// TIA Portal project "Supervisorios2" (V17)

(* hardware
DEVICE "S7-1200 station_1"  S7-1200 Station
   slot 0: "Rack_0"  S7-1200 Rack  Rack  V1.0
   slot 1: "PLC_1"  CPU 1212C AC/DC/Rly  6ES7 212-1BE40-0XB0  V4.4
   slot 2: "DI 8x24VDC_1"  6ES7 221-1BF32-0XB0  V2.0
   slot 3: "AQ 1x12BIT_1"  AQ1 signal board  6ES7 232-4HA30-0XB0  V1.0
DEVICE "HMI_1"  TP700 Comfort
   slot 0: "HMI_1"  TP700 Comfort  6AV2 124-0GC01-0AX0  17.0.0.0
   slot 1: "HMI_RT_1"  TP700 Comfort  6AV2 124-0GC01-0AX0  17.0.0.0
   slot 5: "HMI_1.IE_CP_1"  PROFINET Interface  17.0.0.0
      slot 1: "PROFINET Interface_1"  PROFINET Interface
         slot 1: "Port_1"  Port
         slot 2: "Port_2"  Port
   slot 7: "HMI_1.MPI/DP_CP_1"  MPI/DP Interface  17.0.0.0
*)

// ===== PLC "PLC_1"  CPU 1212C AC/DC/Rly =====

VAR_GLOBAL   // PLC tag table "Default tag table"
   "MemLED" AT %M32.0 : Bool;
   "MemL" AT %M32.1 : Bool;
   "norm" AT %MD8 : Real;
   "scal" AT %MD12 : Real;
   "potenciometro" AT %IW64 : Word;
   "SAIDA" AT %QD2 : Real;
   "Tag_2" AT %M101.2 : Bool;
   "Clock_Byte" AT %MB0 : Byte;
   "Clock_10Hz" AT %M0.0 : Bool;
   "Clock_5Hz" AT %M0.1 : Bool;
   "Clock_2.5Hz" AT %M0.2 : Bool;
   "Clock_2Hz" AT %M0.3 : Bool;
   "Clock_1.25Hz" AT %M0.4 : Bool;
   "Clock_1Hz" AT %M0.5 : Bool;
   "Clock_0.625Hz" AT %M0.6 : Bool;
   "Clock_0.5Hz" AT %M0.7 : Bool;
END_VAR

VAR_GLOBAL   // PLC tag table "ComportamentoRipas"
   "ON" AT %I0.0 : Bool;
   "OFF" AT %I0.1 : Bool;
   "S1" AT %I0.2 : Bool;
   "S2" AT %I0.3 : Bool;
   "A" AT %I0.4 : Bool;
   "O" AT %I0.5 : Bool;
   "P" AT %I0.6 : Bool;
   "L" AT %I0.7 : Bool;
   "M" AT %I8.0 : Bool;
   "N" AT %I8.1 : Bool;
   "MA" AT %Q0.0 : Bool;
   "MS" AT %Q0.1 : Bool;
   "ME" AT %Q0.2 : Bool;
   "C1" AT %Q0.3 : Bool;
   "C2" AT %Q0.4 : Bool;
   "Estado0" AT %M100.0 : Bool;
   "Estado1" AT %M100.1 : Bool;
   "Estado2" AT %M100.2 : Bool;
   "Estado3" AT %M100.3 : Bool;
   "Estado4" AT %M100.4 : Bool;
   "Estado5" AT %M100.5 : Bool;
   "Estado6" AT %M100.6 : Bool;
   "Estado7" AT %M100.7 : Bool;
   "MemOFF" AT %M101.1 : Bool;
   "Estado8" AT %M101.0 : Bool;
   "LedTeste" AT %Q0.5 : Bool;
END_VAR

TYPE "Receita"
   STRUCT
      ComprimentoRipa : Real;
      OutroTipo : UInt;
   END_STRUCT;
END_TYPE

TYPE "DT_Cilindro"
   STRUCT
      NomeCilindro : String;
      EstadoCilindro : Bool;
      EstadoSensorMin : Bool;
      EstadoSensorMax : Bool;
      ModoControle : Bool;
      ComprimentoXEixo : Int;
      VelocidadeEixo : Int;
   END_STRUCT;
END_TYPE

DATA_BLOCK "Dados_IHM"   // DB1
{ S7_Optimized_Access := 'TRUE' }
VERSION : 0.1
   VAR
      IHM_Screen : Array[0..4] of UInt;
      LED : Bool;
      Botão : Bool;
      SetaTela : UInt := 4;
      POT : Real;
   END_VAR
BEGIN
END_DATA_BLOCK

DATA_BLOCK "Alarmes"   // DB2
{ S7_Optimized_Access := 'FALSE' }
VERSION : 0.1
   VAR
      ALARME : Array[0..1] of Word;
      ALARMEAnalog : Word;
   END_VAR
BEGIN
END_DATA_BLOCK

DATA_BLOCK "Receita_IHM"   // DB3
{ S7_Optimized_Access := 'FALSE' }
VERSION : 0.1
   VAR
      ComprimentoRipa : Real;
      OutroElemento : UInt;
      NomeReceita : WString;
      ReceitasCustom : Array[0..3] of "Receita";
      Atual : "Receita";
      UltimoCarregado : Byte;
      RetMOVBLK : Int;
      BoolCarregado : Bool;
   END_VAR
BEGIN
END_DATA_BLOCK

DATA_BLOCK "DB_Cilindro"   // DB4
{ S7_Optimized_Access := 'TRUE' }
VERSION : 0.1
   VAR RETAIN
      Cilindro1 : "DT_Cilindro";
      Cilindro2 : "DT_Cilindro";
   END_VAR
BEGIN
   Cilindro1.NomeCilindro := 'pistao um';
   Cilindro1.EstadoSensorMin := true;
   Cilindro2.NomeCilindro := 'pistao dois';
   Cilindro2.EstadoSensorMin := true;
   Cilindro1.VelocidadeEixo := 15;
   Cilindro2.VelocidadeEixo := 25;
END_DATA_BLOCK

DATA_BLOCK "ControleCilindro_DB"   // DB5
{ S7_Optimized_Access := 'TRUE' }
VERSION : 0.1
// stored: InstanceOfName ControleCilindro
"ControleCilindro"
BEGIN
END_DATA_BLOCK

FUNCTION_BLOCK "ControleCilindro"   // FB1, LAD
{ S7_Optimized_Access := 'TRUE' }
VERSION : 0.1
   VAR_IN_OUT
      Cilindro : "DT_Cilindro";
   END_VAR
   VAR_TEMP
      ComprimentoModif : Int;
   END_VAR
   VAR_TEMP   // added for the SCL form of the ladder/FBD networks
      _w1 : Bool;
   END_VAR
BEGIN

REGION Network 1
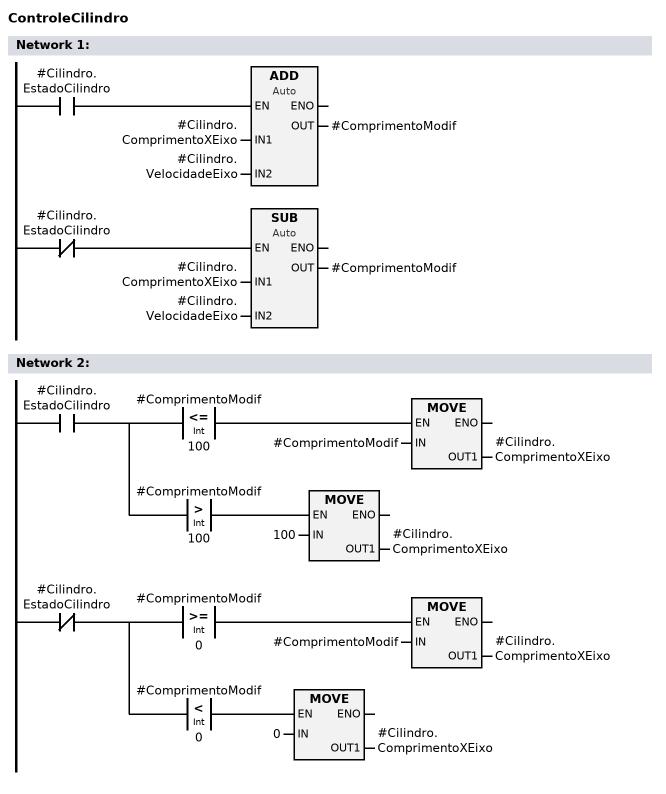
   RUNG wire#powerrail
      Contact( #Cilindro.EstadoCilindro )
      Add(in1 := #Cilindro.ComprimentoXEixo, in2 := #Cilindro.VelocidadeEixo, out => #ComprimentoModif)
   END_RUNG
   RUNG wire#powerrail
      I_Contact( #Cilindro.EstadoCilindro )
      Sub(in1 := #Cilindro.ComprimentoXEixo, in2 := #Cilindro.VelocidadeEixo, out => #ComprimentoModif)
   END_RUNG
   // the same network as SCL:
   IF #Cilindro.EstadoCilindro THEN
       #ComprimentoModif := #Cilindro.ComprimentoXEixo + #Cilindro.VelocidadeEixo;
   END_IF;
   IF NOT #Cilindro.EstadoCilindro THEN
       #ComprimentoModif := #Cilindro.ComprimentoXEixo - #Cilindro.VelocidadeEixo;
   END_IF;
END_REGION

REGION Network 2
   RUNG wire#powerrail
      Contact( #Cilindro.EstadoCilindro )
      wire#w1
      { S7_Templates := "SrcType := Int" } LE_Contact(in1 := #ComprimentoModif, in2 := 100)
      Move(in := #ComprimentoModif, out1 => #Cilindro.ComprimentoXEixo)
   END_RUNG
   RUNG wire#w1
      { S7_Templates := "SrcType := Int" } GT_Contact(in1 := #ComprimentoModif, in2 := 100)
      Move(in := 100, out1 => #Cilindro.ComprimentoXEixo)
   END_RUNG
   RUNG wire#powerrail
      I_Contact( #Cilindro.EstadoCilindro )
      wire#w2
      { S7_Templates := "SrcType := Int" } GE_Contact(in1 := #ComprimentoModif, in2 := 0)
      Move(in := #ComprimentoModif, out1 => #Cilindro.ComprimentoXEixo)
   END_RUNG
   RUNG wire#w2
      { S7_Templates := "SrcType := Int" } LT_Contact(in1 := #ComprimentoModif, in2 := 0)
      Move(in := 0, out1 => #Cilindro.ComprimentoXEixo)
   END_RUNG
   // the same network as SCL:
   IF #Cilindro.EstadoCilindro AND (#ComprimentoModif <= 100) THEN
       #Cilindro.ComprimentoXEixo := #ComprimentoModif;
   END_IF;
   IF #Cilindro.EstadoCilindro AND (#ComprimentoModif > 100) THEN #Cilindro.ComprimentoXEixo := 100; END_IF;
   #_w1 := NOT #Cilindro.EstadoCilindro;
   IF #_w1 AND (#ComprimentoModif >= 0) THEN #Cilindro.ComprimentoXEixo := #ComprimentoModif; END_IF;
   IF #_w1 AND (#ComprimentoModif < 0) THEN #Cilindro.ComprimentoXEixo := 0; END_IF;
END_REGION
END_FUNCTION_BLOCK

ORGANIZATION_BLOCK "Main"   // OB1, LAD, ProgramCycle
TITLE = "Main Program Sweep (Cycle)"
{ S7_Optimized_Access := 'TRUE' }
VERSION : 0.1
   VAR_INPUT
      Initial_Call : Bool;   // Initial call of this OB
      Remanence : Bool;   // =True, if remanent data are available
   END_VAR
   VAR_TEMP   // added for the SCL form of the ladder/FBD networks
      _w1 : Bool;
   END_VAR
BEGIN

REGION Network 1: Estado Inicial
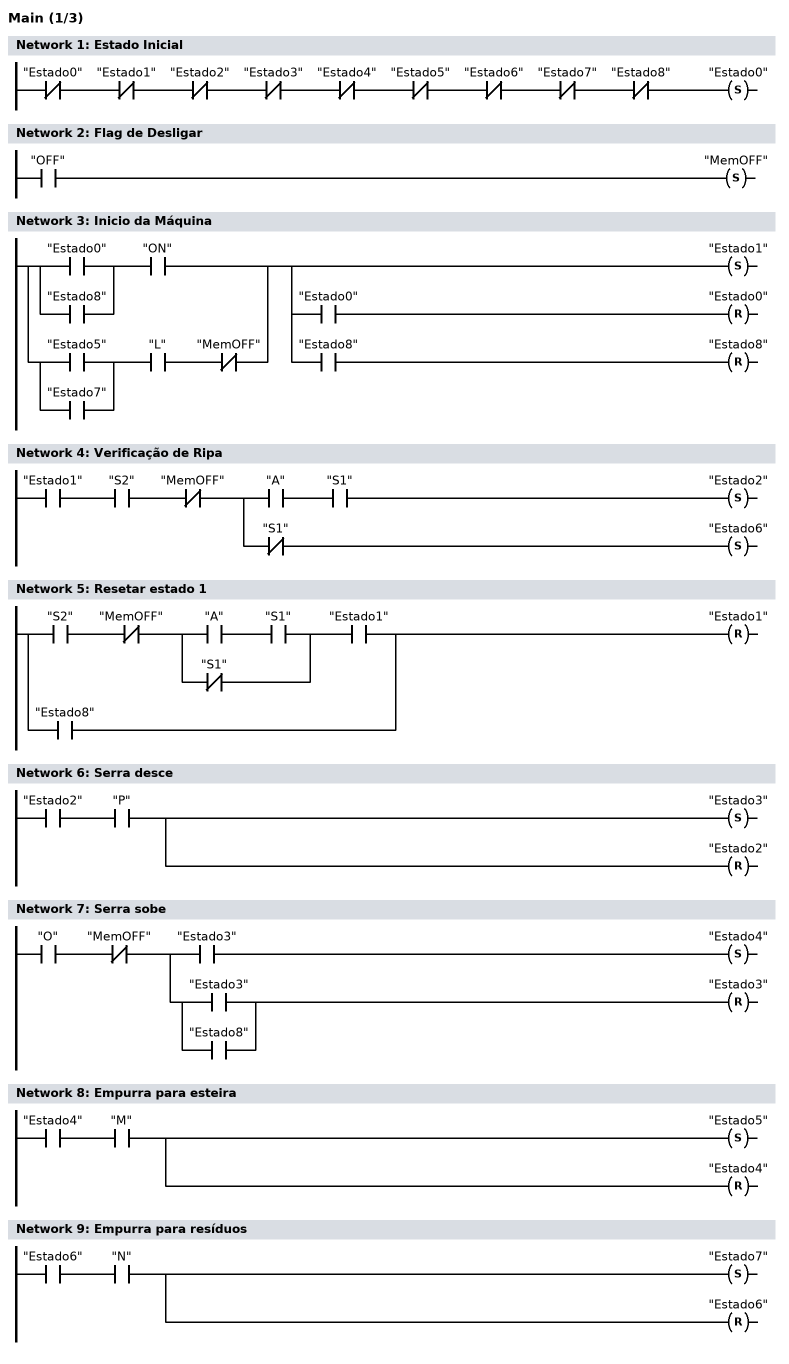
   RUNG wire#powerrail
      I_Contact( "Estado0" )
      I_Contact( "Estado1" )
      I_Contact( "Estado2" )
      I_Contact( "Estado3" )
      I_Contact( "Estado4" )
      I_Contact( "Estado5" )
      I_Contact( "Estado6" )
      I_Contact( "Estado7" )
      I_Contact( "Estado8" )
      S_Coil( "Estado0" )
   END_RUNG
   // the same network as SCL:
   IF NOT "Estado0" AND NOT "Estado1" AND NOT "Estado2" AND NOT "Estado3" AND NOT "Estado4" AND NOT "Estado5" AND NOT "Estado6" AND NOT "Estado7" AND NOT "Estado8" THEN
       "Estado0" := TRUE;
   END_IF;
END_REGION

REGION Network 2: Flag de Desligar
   RUNG wire#powerrail
      Contact( "OFF" )
      S_Coil( "MemOFF" )
   END_RUNG
   // the same network as SCL:
   IF "OFF" THEN "MemOFF" := TRUE; END_IF;
END_REGION

REGION Network 3: Inicio da Máquina
   RUNG wire#powerrail
      Contact( "Estado0" )
      wire#w1
      Contact( "ON" )
      wire#w2
      S_Coil( "Estado1" )
   END_RUNG
   RUNG wire#powerrail
      Contact( "Estado8" )
   END_RUNG wire#w1
   RUNG wire#powerrail
      Contact( "Estado5" )
      wire#w3
      Contact( "L" )
      I_Contact( "MemOFF" )
   END_RUNG wire#w2
   RUNG wire#powerrail
      Contact( "Estado7" )
   END_RUNG wire#w3
   RUNG wire#w2
      Contact( "Estado0" )
      R_Coil( "Estado0" )
   END_RUNG
   RUNG wire#w2
      Contact( "Estado8" )
      R_Coil( "Estado8" )
   END_RUNG
   // the same network as SCL:
   #_w1 := (("Estado0" OR "Estado8") AND "ON") OR (("Estado5" OR "Estado7") AND "L" AND NOT "MemOFF");
   IF #_w1 THEN "Estado1" := TRUE; END_IF;
   IF #_w1 AND "Estado0" THEN "Estado0" := FALSE; END_IF;
   IF #_w1 AND "Estado8" THEN "Estado8" := FALSE; END_IF;
END_REGION

REGION Network 4: Verificação de Ripa
   RUNG wire#powerrail
      Contact( "Estado1" )
      Contact( "S2" )
      I_Contact( "MemOFF" )
      wire#w1
      Contact( "A" )
      Contact( "S1" )
      S_Coil( "Estado2" )
   END_RUNG
   RUNG wire#w1
      I_Contact( "S1" )
      S_Coil( "Estado6" )
   END_RUNG
   // the same network as SCL:
   #_w1 := "Estado1" AND "S2" AND NOT "MemOFF";
   IF #_w1 AND "A" AND "S1" THEN "Estado2" := TRUE; END_IF;
   IF #_w1 AND NOT "S1" THEN "Estado6" := TRUE; END_IF;
END_REGION

REGION Network 5: Resetar estado 1
   RUNG wire#powerrail
      Contact( "S2" )
      I_Contact( "MemOFF" )
      wire#w1
      Contact( "A" )
      Contact( "S1" )
      wire#w2
      Contact( "Estado1" )
      wire#w3
      R_Coil( "Estado1" )
   END_RUNG
   RUNG wire#w1
      I_Contact( "S1" )
   END_RUNG wire#w2
   RUNG wire#powerrail
      Contact( "Estado8" )
   END_RUNG wire#w3
   // the same network as SCL:
   IF ("S2" AND NOT "MemOFF" AND (("A" AND "S1") OR NOT "S1") AND "Estado1") OR "Estado8" THEN
       "Estado1" := FALSE;
   END_IF;
END_REGION

REGION Network 6: Serra desce
   RUNG wire#powerrail
      Contact( "Estado2" )
      Contact( "P" )
      wire#w1
      S_Coil( "Estado3" )
   END_RUNG
   RUNG wire#w1
      R_Coil( "Estado2" )
   END_RUNG
   // the same network as SCL:
   IF "Estado2" AND "P" THEN
       "Estado3" := TRUE;
       "Estado2" := FALSE;
   END_IF;
END_REGION

REGION Network 7: Serra sobe
   RUNG wire#powerrail
      Contact( "O" )
      I_Contact( "MemOFF" )
      wire#w1
      Contact( "Estado3" )
      S_Coil( "Estado4" )
   END_RUNG
   RUNG wire#w1
      Contact( "Estado3" )
      wire#w2
      R_Coil( "Estado3" )
   END_RUNG
   RUNG wire#w1
      Contact( "Estado8" )
   END_RUNG wire#w2
   // the same network as SCL:
   #_w1 := "O" AND NOT "MemOFF";
   IF #_w1 AND "Estado3" THEN "Estado4" := TRUE; END_IF;
   IF #_w1 AND ("Estado3" OR "Estado8") THEN "Estado3" := FALSE; END_IF;
END_REGION

REGION Network 8: Empurra para esteira
   RUNG wire#powerrail
      Contact( "Estado4" )
      Contact( "M" )
      wire#w1
      S_Coil( "Estado5" )
   END_RUNG
   RUNG wire#w1
      R_Coil( "Estado4" )
   END_RUNG
   // the same network as SCL:
   IF "Estado4" AND "M" THEN
       "Estado5" := TRUE;
       "Estado4" := FALSE;
   END_IF;
END_REGION

REGION Network 9: Empurra para resíduos
   RUNG wire#powerrail
      Contact( "Estado6" )
      Contact( "N" )
      wire#w1
      S_Coil( "Estado7" )
   END_RUNG
   RUNG wire#w1
      R_Coil( "Estado6" )
   END_RUNG
   // the same network as SCL:
   IF "Estado6" AND "N" THEN
       "Estado7" := TRUE;
       "Estado6" := FALSE;
   END_IF;
END_REGION

REGION Network 10: Recua para posição inicial
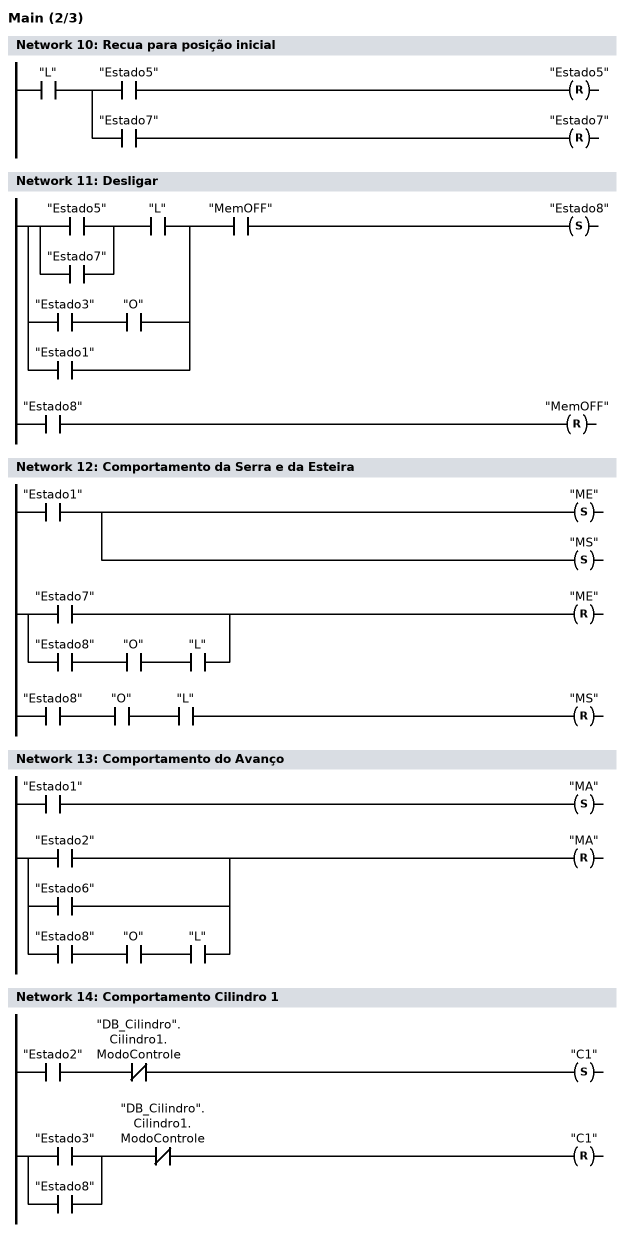
   RUNG wire#powerrail
      Contact( "L" )
      wire#w1
      Contact( "Estado5" )
      R_Coil( "Estado5" )
   END_RUNG
   RUNG wire#w1
      Contact( "Estado7" )
      R_Coil( "Estado7" )
   END_RUNG
   // the same network as SCL:
   IF "L" AND "Estado5" THEN "Estado5" := FALSE; END_IF;
   IF "L" AND "Estado7" THEN "Estado7" := FALSE; END_IF;
END_REGION

REGION Network 11: Desligar
   RUNG wire#powerrail
      Contact( "Estado5" )
      wire#w1
      Contact( "L" )
      wire#w2
      Contact( "MemOFF" )
      S_Coil( "Estado8" )
   END_RUNG
   RUNG wire#powerrail
      Contact( "Estado7" )
   END_RUNG wire#w1
   RUNG wire#powerrail
      Contact( "Estado3" )
      Contact( "O" )
   END_RUNG wire#w2
   RUNG wire#powerrail
      Contact( "Estado1" )
   END_RUNG wire#w2
   RUNG wire#powerrail
      Contact( "Estado8" )
      R_Coil( "MemOFF" )
   END_RUNG
   // the same network as SCL:
   IF ((("Estado5" OR "Estado7") AND "L") OR ("Estado3" AND "O") OR "Estado1") AND "MemOFF" THEN
       "Estado8" := TRUE;
   END_IF;
   IF "Estado8" THEN "MemOFF" := FALSE; END_IF;
END_REGION

REGION Network 12: Comportamento da Serra e da Esteira
   RUNG wire#powerrail
      Contact( "Estado1" )
      wire#w1
      S_Coil( "ME" )
   END_RUNG
   RUNG wire#w1
      S_Coil( "MS" )
   END_RUNG
   RUNG wire#powerrail
      Contact( "Estado7" )
      wire#w2
      R_Coil( "ME" )
   END_RUNG
   RUNG wire#powerrail
      Contact( "Estado8" )
      Contact( "O" )
      Contact( "L" )
   END_RUNG wire#w2
   RUNG wire#powerrail
      Contact( "Estado8" )
      Contact( "O" )
      Contact( "L" )
      R_Coil( "MS" )
   END_RUNG
   // the same network as SCL:
   IF "Estado1" THEN
       "ME" := TRUE;
       "MS" := TRUE;
   END_IF;
   IF "Estado7" OR ("Estado8" AND "O" AND "L") THEN "ME" := FALSE; END_IF;
   IF "Estado8" AND "O" AND "L" THEN "MS" := FALSE; END_IF;
END_REGION

REGION Network 13: Comportamento do Avanço
   RUNG wire#powerrail
      Contact( "Estado1" )
      S_Coil( "MA" )
   END_RUNG
   RUNG wire#powerrail
      Contact( "Estado2" )
      wire#w1
      R_Coil( "MA" )
   END_RUNG
   RUNG wire#powerrail
      Contact( "Estado6" )
   END_RUNG wire#w1
   RUNG wire#powerrail
      Contact( "Estado8" )
      Contact( "O" )
      Contact( "L" )
   END_RUNG wire#w1
   // the same network as SCL:
   IF "Estado1" THEN "MA" := TRUE; END_IF;
   IF "Estado2" OR "Estado6" OR ("Estado8" AND "O" AND "L") THEN "MA" := FALSE; END_IF;
END_REGION

REGION Network 14: Comportamento Cilindro 1
   RUNG wire#powerrail
      Contact( "Estado2" )
      I_Contact( "DB_Cilindro".Cilindro1.ModoControle )
      S_Coil( "C1" )
   END_RUNG
   RUNG wire#powerrail
      Contact( "Estado3" )
      wire#w1
      I_Contact( "DB_Cilindro".Cilindro1.ModoControle )
      R_Coil( "C1" )
   END_RUNG
   RUNG wire#powerrail
      Contact( "Estado8" )
   END_RUNG wire#w1
   // the same network as SCL:
   IF "Estado2" AND NOT "DB_Cilindro".Cilindro1.ModoControle THEN "C1" := TRUE; END_IF;
   IF ("Estado3" OR "Estado8") AND NOT "DB_Cilindro".Cilindro1.ModoControle THEN "C1" := FALSE; END_IF;
END_REGION

REGION Network 15: Comportamento Cilindro 2
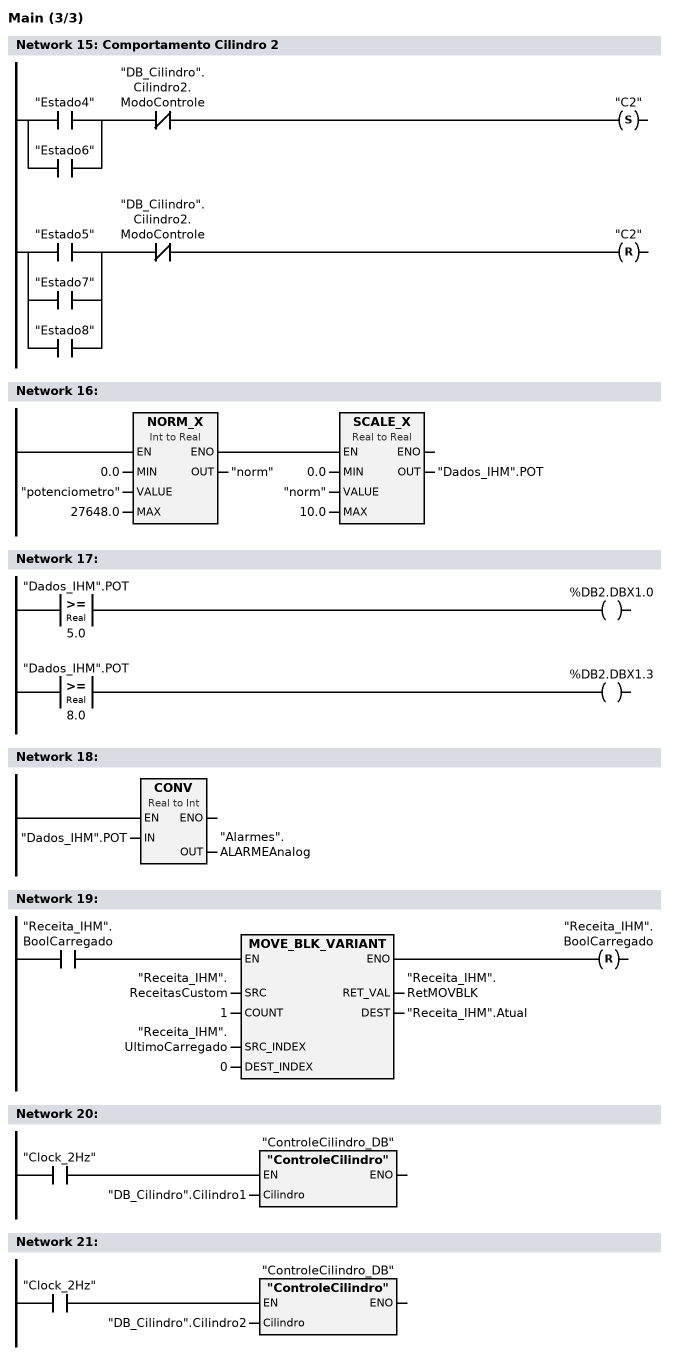
   RUNG wire#powerrail
      Contact( "Estado4" )
      wire#w1
      I_Contact( "DB_Cilindro".Cilindro2.ModoControle )
      S_Coil( "C2" )
   END_RUNG
   RUNG wire#powerrail
      Contact( "Estado6" )
   END_RUNG wire#w1
   RUNG wire#powerrail
      Contact( "Estado5" )
      wire#w2
      I_Contact( "DB_Cilindro".Cilindro2.ModoControle )
      R_Coil( "C2" )
   END_RUNG
   RUNG wire#powerrail
      Contact( "Estado7" )
   END_RUNG wire#w2
   RUNG wire#powerrail
      Contact( "Estado8" )
   END_RUNG wire#w2
   // the same network as SCL:
   IF ("Estado4" OR "Estado6") AND NOT "DB_Cilindro".Cilindro2.ModoControle THEN "C2" := TRUE; END_IF;
   IF ("Estado5" OR "Estado7" OR "Estado8") AND NOT "DB_Cilindro".Cilindro2.ModoControle THEN
       "C2" := FALSE;
   END_IF;
END_REGION

REGION Network 16
   RUNG wire#powerrail
      { S7_Templates := "[SrcType := Int, DestType := Real]" } Normalize(min := 0.0, value := "potenciometro", max := 27648.0, out => "norm")
      { S7_Templates := "[SrcType := Real, DestType := Real]" } Scale(min := 0.0, value := "norm", max := 10.0, out => "Dados_IHM".POT)
   END_RUNG
   // the same network as SCL:
   "norm" := NORM_X(MIN := 0.0, VALUE := "potenciometro", MAX := 27648.0);
   "Dados_IHM".POT := SCALE_X(MIN := 0.0, VALUE := "norm", MAX := 10.0);
END_REGION

REGION Network 17
   RUNG wire#powerrail
      { S7_Templates := "SrcType := Real" } GE_Contact(in1 := "Dados_IHM".POT, in2 := 5.0)
      Coil( %DB2.DBX1.0 )
   END_RUNG
   RUNG wire#powerrail
      { S7_Templates := "SrcType := Real" } GE_Contact(in1 := "Dados_IHM".POT, in2 := 8.0)
      Coil( %DB2.DBX1.3 )
   END_RUNG
   // the same network as SCL:
   %DB2.DBX1.0 := "Dados_IHM".POT >= 5.0;
   %DB2.DBX1.3 := "Dados_IHM".POT >= 8.0;
END_REGION

REGION Network 18
   RUNG wire#powerrail
      { S7_Templates := "[SrcType := Real, DestType := Int]" } Convert(in := "Dados_IHM".POT, out => "Alarmes".ALARMEAnalog)
   END_RUNG
   // the same network as SCL:
   "Alarmes".ALARMEAnalog := REAL_TO_INT("Dados_IHM".POT);
END_REGION

REGION Network 19
   // ENO of a box is taken as its EN; it also drops when the box reports an error
   #_w1 := "Receita_IHM".BoolCarregado;
   IF #_w1 THEN
       "Receita_IHM".RetMOVBLK := MOVE_BLK_VARIANT(SRC := "Receita_IHM".ReceitasCustom,
                               COUNT := 1,
                               SRC_INDEX := "Receita_IHM".UltimoCarregado,
                               DEST_INDEX := 0,
                               DEST => "Receita_IHM".Atual);
       "Receita_IHM".BoolCarregado := FALSE;
   END_IF;
END_REGION

REGION Network 20
   RUNG wire#powerrail
      Contact( "Clock_2Hz" )
      "ControleCilindro_DB"(Cilindro := "DB_Cilindro".Cilindro1)
   END_RUNG
   // the same network as SCL:
   IF "Clock_2Hz" THEN
       "ControleCilindro_DB"(Cilindro := "DB_Cilindro".Cilindro1);   // "ControleCilindro"
   END_IF;
END_REGION

REGION Network 21
   RUNG wire#powerrail
      Contact( "Clock_2Hz" )
      "ControleCilindro_DB"(Cilindro := "DB_Cilindro".Cilindro2)
   END_RUNG
   // the same network as SCL:
   IF "Clock_2Hz" THEN
       "ControleCilindro_DB"(Cilindro := "DB_Cilindro".Cilindro2);   // "ControleCilindro"
   END_IF;
END_REGION
END_ORGANIZATION_BLOCK

(* ===== HMI "HMI_RT_1" =====
system functions are stored by id; their names below are inferred from use
connection "HMI_Connection_1": ETHERNET, S7_1200_OMS

HMI tags "Default tag table"
   "Tag_ScreenNumber" : UInt, internal
   "NumeroTela" : UInt = PLC Dados_IHM.SetaTela AT %DB1.DBW0, 500 ms
      on ChangeValue: ActivateScreenByNumber("NumeroTela", 0)
   "LED" : Bool = PLC Dados_IHM.LED AT %DB1.DBX0.0, 1 s
   "Botao" : Bool = PLC Dados_IHM.Botão AT %DB1.DBX0.0, 1 s
   "potenciometro" : Real = PLC Dados_IHM.POT AT %QD2, 1 s
   "pot2" : Word = PLC potenciometro AT %IW64, 1 s
   "usuario" : WString[254] AT %DB1.DBX0.0
   "grupo" : Int AT %DB1.DBW0
   "Alarmes_ALARME" : Array [0..1] of Word = PLC Alarmes.ALARME AT %DB2.DBX0.0, 1 s
   "Alarmes_ALARMEAnalog" : Word = PLC Alarmes.ALARMEAnalog AT %DB2.DBW4, 1 s
   "Receita_IHM_ComprimentoRipa" : Real = PLC Receita_IHM.ComprimentoRipa AT %DB3.DBD0, 1 s
   "Receita_IHM_OutroElemento" : UInt = PLC Receita_IHM.OutroElemento AT %DB3.DBW4, 1 s
   "Receita_IHM_NomeReceita" : WString[254] = PLC Receita_IHM.NomeReceita AT %DB3.DBX6.0, 1 s
   "NomeReceita" : WString[254], internal
   "usuario_1" : WString[254], internal
   "Receita_IHM_ReceitasCustom{0}_ComprimentoRipa" : Real = PLC Receita_IHM.ReceitasCustom[0].ComprimentoRipa AT %DB3.DBD518, 1 s
   "Receita_IHM_ReceitasCustom{0}_OutroTipo" : UInt = PLC Receita_IHM.ReceitasCustom[0].OutroTipo AT %DB3.DBW522, 1 s
   "Receita_IHM_ReceitasCustom{1}_ComprimentoRipa" : Real = PLC Receita_IHM.ReceitasCustom[1].ComprimentoRipa AT %DB3.DBD524, 1 s
   "Receita_IHM_ReceitasCustom{1}_OutroTipo" : UInt = PLC Receita_IHM.ReceitasCustom[1].OutroTipo AT %DB3.DBW528, 1 s
   "Receita_IHM_Atual_ComprimentoRipa" : Real = PLC Receita_IHM.Atual.ComprimentoRipa AT %DB3.DBD542, 1 s
   "Receita_IHM_Atual_OutroTipo" : UInt = PLC Receita_IHM.Atual.OutroTipo AT %DB3.DBW546, 1 s
   "Receita_IHM_BoolCarregado" : Bool = PLC Receita_IHM.BoolCarregado AT %DB3.DBX552.0, 1 s
   "Receita_IHM_UltimoCarregado" : Byte = PLC Receita_IHM.UltimoCarregado AT %DB3.DBB548, 1 s
   "Receita_IHM_ReceitasCustom{2}_ComprimentoRipa" : Real = PLC Receita_IHM.ReceitasCustom[2].ComprimentoRipa AT %DB3.DBD530, 1 s
   "Receita_IHM_ReceitasCustom{2}_OutroTipo" : UInt = PLC Receita_IHM.ReceitasCustom[2].OutroTipo AT %DB3.DBW534, 1 s
   "Receita_IHM_ReceitasCustom{3}_ComprimentoRipa" : Real = PLC Receita_IHM.ReceitasCustom[3].ComprimentoRipa AT %DB3.DBD536, 1 s
   "Receita_IHM_ReceitasCustom{3}_OutroTipo" : UInt = PLC Receita_IHM.ReceitasCustom[3].OutroTipo AT %DB3.DBW540, 1 s

HMI tags "Tags_Cilindro"
   "DB_Cilindro_Cilindro1" : DT_Cilindro = PLC DB_Cilindro.Cilindro1, 1 s
   "DB_Cilindro_Cilindro2" : DT_Cilindro = PLC DB_Cilindro.Cilindro2, 1 s

discrete alarms
   1: 'Ripa Ausente / AAAAAAAAAA', class Warnings, trigger "Alarmes_ALARME" bit 0
   2: 'Motor Serra Desligado', class Warnings, trigger "Alarmes_ALARME" bit 1
   3: 'Motor Esteira Parado', class Warnings, trigger "Alarmes_ALARME" bit 2
   4: 'Sensores com Defeito', class Errors, trigger "Alarmes_ALARME" bit 3
   5: 'Multiplos Estados Ativos', class Errors, trigger "Alarmes_ALARME" bit 4

analog alarms
   2: 'Comprimento Ripa abaixo da norma', class Errors, trigger "Alarmes_ALARMEAnalog"
   3: 'Velocidade de entrada de ripas abaixo do esperado', class Warnings, trigger "Alarmes_ALARMEAnalog"
   4: 'Velocidade de entrada de ripas acima do esperado', class Errors, trigger "Alarmes_ALARMEAnalog"
   5: 'Multiplas Ripas defeituosas', class Warnings, trigger "Alarmes_ALARMEAnalog"
   1: 'Comprimento Ripa acima da norma', class Errors, trigger "Alarmes_ALARMEAnalog"

text list "On_Off": 0 'Off'; 1 'On'

graphic list "ONOFF": 0 'Graphic_3'; 1 'Graphic_2'

recipe "PadraoRipa": ComprimentoRipa <- "Receita_IHM_ComprimentoRipa", OutroElemento <- "Receita_IHM_OutroElemento"

SlideinScreen "GraphX_Slidein_Left" 267x480
   Button "Button_1" at 32,209 size 192x32; TextOff 'Pop-up screen_1'
      on Click: function_cf6f4242("GraphX_Slidein_Left", 1)

screen "DELETARLogin" 800x420
   on GenerateScreen: SetTag("Tag_ScreenNumber", 1)
   TextField "HmiScreenItemData_4" at 0,2 size 576x25; Text 'Welcome to HMI_1 (TP700 Comfort)!'
   Button "HmiScreenItemData" at 36,36 size 159x47; TextOff 'Screen0'; PictureOff "Navigates to Screen0 for TP700 Comfort 17.0.0.0"; PictureOn "Navigates to Screen0 for TP700 Comfort 17.0.0.0"
      on Release: ActivateScreen("DELETARTopologia", 0)
   Button "HmiScreenItemData_1" at 36,95 size 159x47; TextOff 'Screen1'; PictureOff "Navigates to Screen1 for TP700 Comfort 17.0.0.0"; PictureOn "Navigates to Screen1 for TP700 Comfort 17.0.0.0"
      on Release: ActivateScreen("DELETARConfiguracao", 0)
   Button "HmiScreenItemData_2" at 36,154 size 159x47; TextOff 'Screen2'; PictureOff "Navigates to Screen2 for TP700 Comfort 17.0.0.0"; PictureOn "Navigates to Screen2 for TP700 Comfort 17.0.0.0"
      on Release: ActivateScreen("DELETARRelatorio", 0)
   Button "HmiScreenItemData_3" at 36,213 size 159x47; TextOff 'Screen3'; PictureOff "Navigates to Screen3 for TP700 Comfort 17.0.0.0"; PictureOn "Navigates to Screen3 for TP700 Comfort 17.0.0.0"
      on Release: ActivateScreen("DELETARAlarmes", 0)
   Button "Button_1" at 718,205 size 77x42; TextOff 'Toggle Led'; TextOn 'Toggling'; TextList "On_Off"; PictureList "ONOFF"
      on Release: InvertBit("Botao")
      ProcessValue <- "Botao"
   IOField "I/O field_1" at 621,110 size 96x32; FormatPattern 1
      ProcessValue <- "LED"
   SymbolicIOField "Symbolic I/O field_1" at 609,148 size 170x32; TextOff '0'; TextOn '1'; TextList "On_Off"
      ProcessValue <- "Botao"
   GraphicIOField "Graphic I/O field_1" at 718,256 size 61x45; PictureList "ONOFF"
      ProcessValue <- "Botao"
   Button "Button_2" at 453,342 size 220x40; TextOff 'Pop-Up Description / Descrição de Pop-Up / Descricíon de Pop-Up'
      on Click: function_cf6f4242("GraphX_Slidein_Left", -1)
   Bar "Bar_1" at 519,58 size 80x230; MinimumValue 0; MaximumValue 10
      ProcessValue <- "potenciometro"
   Button "Button_3" at 239,81 size 145x48; TextOff 'login / conectar / iniciar sesión'
      on Click: function_a2a04561()
   Button "Button_4" at 234,149 size 147x56; TextOff 'logout / desconectar / cerrar sesión'
      on Click: function_f23ef4c9()
   IOField "I/O field_2" at 339,213 size 169x62; FormatPattern ??????????
      ProcessValue <- "usuario"
   Button "Button_5" at 406,117 size 107x55; TextOff 'confirm / confirmar'; Authorization "Monitor"
      on Click: function_f41c6f6c("usuario")
   Button "Button_6" at 67,320 size 98x61; TextOff 'Text'; PictureOff "Graphic_2"
      on Release: function_fb9197e8(L pt-BR)
   Button "Button_7" at 183,320 size 95x61; TextOff 'Text'; PictureOff "Graphic_5"
      on Release: function_fb9197e8(L en-US)
   Button "Button_8" at 293,320 size 104x61; TextOff 'Text'; PictureOff "Graphic_6"
      on Release: function_fb9197e8(L es-ES)
   Button "HmiScreenItemData_5" at 32,273 size 159x47; TextOn 'Screen3'; TextOff 'Carregar Receita'; PictureOn "Navigates to Screen3 for TP700 Comfort 17.0.0.0"; PictureOff "Navigates to Screen3 for TP700 Comfort 17.0.0.0"
      on Release: ActivateScreen("DELETARReceita", 0)

Template "Navegação" 800x420
   Button "Alarms" at 235,351 size 78x58; TextOff 'Alarms'; PictureOff "AlarmDisplay_TP700_Comfort_TR"; PictureOn "AlarmDisplay_TP700_Comfort_TR"
      on Release: function_ef3f5d25("Alarm window_Unacknowledged", -1)
   Button "BotaoTopologia" at 42,351 size 78x58; TextOff 'Topologia'
      on Release: ActivateScreen("DELETARTopologia", 0)
   Button "BotaoConfig" at 475,351 size 78x58; TextOff 'Configuração'
      on Release: ActivateScreen("DELETARConfiguracao", 0)
   Button "Template_Button_5" at 720,360 size 78x58; TextOff 'Relatorio'
      on Release: ActivateScreen("DELETARRelatorio", 0)
   Button "BotaoAlarme" at 362,353 size 78x58; TextOff 'Alarme'
      on Release: ActivateScreen("DELETARAlarmes", 0)
   IOField "Template_I/O field_1" at 21,45 size 224x32; FormatPattern ????????????????????????????????????????????????????????????????????????????????
      ProcessValue <- "NomeReceita"

screen "DELETARTopologia" 800x420, template "Navegação"
   on GenerateScreen: SetTag("Tag_ScreenNumber", 2)
   Button "Back" at 1,1 size 159x47; TextOff 'Back'
      on Release: ActivateScreen("DELETARLogin", 0)

screen "DELETARConfiguracao" 800x420, template "Navegação"
   on GenerateScreen: SetTag("Tag_ScreenNumber", 3)
   Circle "Circle_2" at 226,149 size 33x33
      HorizontalMovement <- "pot2"
   Circle "Circle_4" at 367,122 size 33x33
      DiagonalMovement <- "pot2"
      Visibility <- "pot2"
   RecipeView "Recipe view_1" at 544,1 size 236x344; Tag4DataRecord "NomeReceita"; Recipe "PadraoRipa"

screen "DELETARRelatorio" 800x420, template "Navegação"
   on GenerateScreen: SetTag("Tag_ScreenNumber", 4)
   TextField "HmiScreenItemData" at 72,195 size 576x25; Text 'Screen2'
   Button "Back" at 1,1 size 159x47; TextOff 'Back'
      on Release: ActivateScreen("DELETARLogin", 0)
   AlarmView "Alarm view_1" at 37,52 size 678x300

screen "DELETARAlarmes" 800x420, template "Navegação"
   on GenerateScreen: SetTag("Tag_ScreenNumber", 5)
   TextField "HmiScreenItemData" at 72,195 size 576x25; Text 'Screen3'
   Button "Back" at 1,1 size 159x47; TextOff 'Back'
      on Release: ActivateScreen("DELETARLogin", 0)
   AlarmView "Alarm view_1" at 21,23 size 680x300

PopupScreen "Pop-up screen_1" 240x240
   Button "Button_1" at 205,0 size 34x30; TextOff 'X'
      on Click: function_efd93a16()

screen "DELETARReceita" 800x420
   IOField "I/O field_1" at 211,82 size 96x32; FormatPattern 999999999.999
      ProcessValue <- "Receita_IHM_ReceitasCustom{0}_ComprimentoRipa"
   IOField "I/O field_2" at 211,125 size 96x32; FormatPattern 99999
      ProcessValue <- "Receita_IHM_ReceitasCustom{0}_OutroTipo"
   IOField "I/O field_3" at 351,82 size 96x32; FormatPattern 999999999.999
      ProcessValue <- "Receita_IHM_ReceitasCustom{1}_ComprimentoRipa"
   IOField "I/O field_4" at 351,125 size 96x32; FormatPattern 99999
      ProcessValue <- "Receita_IHM_ReceitasCustom{1}_OutroTipo"
   IOField "I/O field_5" at 494,82 size 96x32; FormatPattern 999999999.999
      ProcessValue <- "Receita_IHM_ReceitasCustom{2}_ComprimentoRipa"
   IOField "I/O field_6" at 494,125 size 96x32; FormatPattern 99999
      ProcessValue <- "Receita_IHM_ReceitasCustom{2}_OutroTipo"
   IOField "I/O field_7" at 639,82 size 96x32; FormatPattern 999999999.999
      ProcessValue <- "Receita_IHM_ReceitasCustom{3}_ComprimentoRipa"
   IOField "I/O field_8" at 639,125 size 96x32; FormatPattern 99999
      ProcessValue <- "Receita_IHM_ReceitasCustom{3}_OutroTipo"
   IOField "I/O field_9" at 211,255 size 96x32; FormatPattern s999999999.999
      ProcessValue <- "Receita_IHM_Atual_ComprimentoRipa"
   IOField "I/O field_10" at 211,298 size 96x32; FormatPattern 99999
      ProcessValue <- "Receita_IHM_Atual_OutroTipo"
   TextField "Text field_1" at 220,229 size 54x23; Text 'Atual'
   TextField "Text field_2" at 73,82 size 126x23; Text 'Comprimento'
   TextField "Text field_3" at 77,125 size 110x23; Text 'Outro Valor'
   TextField "Text field_4" at 69,255 size 126x23; Text 'Comprimento'
   TextField "Text field_5" at 73,298 size 110x23; Text 'Outro Valor'
   Button "Button_1" at 211,174 size 96x32; TextOff 'Load 1'
      on Release: SetBit("Receita_IHM_BoolCarregado"); SetTag("Receita_IHM_UltimoCarregado", 0)
   Button "Button_2" at 351,174 size 96x32; TextOff 'Load 2'
      on Release: SetTag("Receita_IHM_UltimoCarregado", 1); SetBit("Receita_IHM_BoolCarregado")
   Button "Button_3" at 494,174 size 96x32; TextOff 'Load 3'
      on Release: SetTag("Receita_IHM_UltimoCarregado", 2); SetBit("Receita_IHM_BoolCarregado")
   Button "Button_4" at 639,174 size 96x32; TextOff 'Load 4'
      on Release: SetTag("Receita_IHM_UltimoCarregado", 3); SetBit("Receita_IHM_BoolCarregado")

screen "Topologia" 800x420, template "TelaDefinitiva"
   ScreenModuleView "pistao_1" at 189,180 size 192x157; ScreenModuleType ""
   ScreenModuleView "pistao_2" at 409,18 size 192x157; ScreenModuleType ""
   ScreenModuleView "motor_1" at 11,18 size 167x137; ScreenModuleType ""
   ScreenModuleView "motor_2" at 205,18 size 167x137; ScreenModuleType ""
   ScreenModuleView "motor_3" at 434,283 size 167x137; ScreenModuleType ""

Template "TelaDefinitiva" 800x420
   Button "btTemplateTopologia" at 650,39 size 129x66; TextOff 'Topologia'
   Button "btTemplateGrafico" at 650,132 size 129x66; TextOff 'Gráficos'
   Button "btTemplateAlarmes" at 650,225 size 129x66; TextOff 'Alarmes'
   Button "btTemplateConfig" at 650,318 size 129x66; TextOff 'Configuração'

scheduled task "Usuario atual"
   on Action: function_f41c6f6c("usuario"); function_e1ab61de("grupo")
*)

(* ===== HMI "HMI_RT_1" =====

ScreenModuleEditorView "pistao" 640x480
   Button "Button_1" at 310,23 size 103x49; TextOff 'Text'
   IOField "I/O field_1" at 130,24 size 124x41; FormatPattern ????
   Button "Button_2" at 91,291 size 92x45; TextOff 'Text'
   Button "Button_3" at 275,290 size 92x45; TextOff 'Text'
*)

(* ===== HMI "HMI_RT_1" =====
system functions are stored by id; their names below are inferred from use

ScreenModuleEditorView "pistao" 640x480
   Button "manual/automatico" at 280,23 size 133x49; TextOn 'MANUAL'; TextOff 'AUTOMATICO'
      ProcessValue <- "Property_1.ModoControle"
      on Click: InvertBit("Property_1.ModoControle")
   Rectangle "braco_1" at 136,132 size 188x37
      Visibility <- "Property_1.EstadoSensorMax"
   Circle "extendido" at 295,217 size 53x53
      Appearance <- "Property_1.EstadoSensorMax"
   Circle "recolhido" at 114,218 size 53x53
      Appearance <- "Property_1.EstadoSensorMin"
   Rectangle "braco_2" at 135,132 size 125x37
      Visibility <- "Property_1.ComprimentoXEixo"
   IOField "nome_pistao" at 31,26 size 124x41; FormatPattern ??????????
      ProcessValue <- "Property_1.NomeCilindro"
   Button "OFF" at 91,291 size 92x45; TextOff 'OFF'
      Appearance <- "Property_1.EstadoCilindro"
      ObjectEnable <- "Property_1.ModoControle"
   Button "ON" at 275,290 size 92x45; TextOff 'ON'
      Appearance <- "Property_1.EstadoCilindro"
      ObjectEnable <- "Property_1.ModoControle"
   Rectangle "braco2_1" at 324,100 size 24x102
      Visibility <- "Property_1.EstadoSensorMax"
   Rectangle "braco2_2" at 261,101 size 24x102
      Visibility <- "Property_1.ComprimentoXEixo"
   Rectangle "braco" at 136,132 size 55x37
      Visibility <- "Property_1.EstadoSensorMin"
   Rectangle "braco2" at 191,100 size 24x102
      Visibility <- "Property_1.EstadoSensorMin"
*)

(* ===== HMI "HMI_RT_1" =====
system functions are stored by id; their names below are inferred from use

ScreenModuleEditorView "pistao" 640x480
   Button "manual/automatico" at 247,23 size 166x49; TextOn 'MANUAL'; TextOff 'AUTOMATICO'
      on Click: InvertBit("Property_1.ModoControle")
      ProcessValue <- "Property_1.ModoControle"
   Rectangle "braco_1" at 136,132 size 188x37
      Visibility <- "Property_1.EstadoSensorMax"
   Circle "extendido" at 295,217 size 53x53
      Appearance <- "Property_1.EstadoSensorMax"
   Circle "recolhido" at 114,218 size 53x53
      Appearance <- "Property_1.EstadoSensorMin"
   Rectangle "braco_2" at 135,132 size 125x37
      Visibility <- "Property_1.ComprimentoXEixo"
   IOField "nome_pistao" at 31,26 size 188x41; FormatPattern ??????????
      ProcessValue <- "Property_1.NomeCilindro"
   Button "OFF" at 91,291 size 92x45; TextOff 'OFF'
      ObjectEnable <- "Property_1.ModoControle"
      Appearance <- "Property_1.EstadoCilindro"
   Button "ON" at 275,290 size 92x45; TextOff 'ON'
      ObjectEnable <- "Property_1.ModoControle"
      Appearance <- "Property_1.EstadoCilindro"
   Rectangle "braco2_1" at 324,100 size 24x102
      Visibility <- "Property_1.EstadoSensorMax"
   Rectangle "braco2_2" at 261,101 size 24x102
      Visibility <- "Property_1.ComprimentoXEixo"
   Rectangle "braco" at 136,132 size 55x37
      Visibility <- "Property_1.EstadoSensorMin"
   Rectangle "braco2" at 191,100 size 24x102
      Visibility <- "Property_1.EstadoSensorMin"
*)

(* ===== HMI "HMI_RT_1" =====
system functions are stored by id; their names below are inferred from use

ScreenModuleEditorView "pistao" 640x480
   Button "manual/automatico" at 247,23 size 166x49; TextOn 'MANUAL'; TextOff 'AUTOMATICO'
      on Click: InvertBit("Property_1.ModoControle")
      ProcessValue <- "Property_1.ModoControle"
   Rectangle "braco_1" at 136,132 size 188x37
      Visibility <- "Property_1.EstadoSensorMax"
   Circle "extendido" at 295,217 size 53x53
      Appearance <- "Property_1.EstadoSensorMax"
   Circle "recolhido" at 114,218 size 53x53
      Appearance <- "Property_1.EstadoSensorMin"
   Rectangle "braco_2" at 135,132 size 125x37
      Visibility <- "Property_1.ComprimentoXEixo"
   IOField "nome_pistao" at 31,26 size 188x41; FormatPattern ??????????
      ProcessValue <- "Property_1.NomeCilindro"
   Button "OFF" at 91,291 size 92x45; TextOff 'OFF'
      ObjectEnable <- "Property_1.ModoControle"
      Appearance <- "Property_1.EstadoCilindro"
   Button "ON" at 275,290 size 92x45; TextOff 'ON'
      ObjectEnable <- "Property_1.ModoControle"
      Appearance <- "Property_1.EstadoCilindro"
   Rectangle "braco2_1" at 324,100 size 24x102
      Visibility <- "Property_1.EstadoSensorMax"
   Rectangle "braco2_2" at 261,101 size 24x102
      Visibility <- "Property_1.ComprimentoXEixo"
   Rectangle "braco" at 136,132 size 55x37
      Visibility <- "Property_1.EstadoSensorMin"
   Rectangle "braco2" at 191,100 size 24x102
      Visibility <- "Property_1.EstadoSensorMin"
*)

(* ===== HMI "HMI_RT_1" =====
system functions are stored by id; their names below are inferred from use

ScreenModuleEditorView "pistao" 640x480
   Button "manual/automatico" at 247,23 size 166x49; TextOn 'MANUAL'; TextOff 'AUTOMATICO'
      on Click: InvertBit("Property_1.ModoControle")
      ProcessValue <- "Property_1.ModoControle"
   Rectangle "braco_1" at 154,132 size 188x37
      Visibility <- "Property_1.EstadoSensorMax"
   Circle "extendido" at 313,217 size 53x53
      Appearance <- "Property_1.EstadoSensorMax"
   Circle "recolhido" at 180,217 size 53x53
      Appearance <- "Property_1.EstadoSensorMin"
   Rectangle "braco_2" at 153,132 size 126x37
      Visibility <- "Property_1.ComprimentoXEixo"
   IOField "nome_pistao" at 31,26 size 188x41; FormatPattern ??????????
      ProcessValue <- "Property_1.NomeCilindro"
   Button "OFF" at 91,291 size 92x45; TextOff 'OFF'
      ObjectEnable <- "Property_1.ModoControle"
      Appearance <- "Property_1.EstadoCilindro"
   Button "ON" at 275,290 size 92x45; TextOff 'ON'
      ObjectEnable <- "Property_1.ModoControle"
      Appearance <- "Property_1.EstadoCilindro"
   Rectangle "braco2_1" at 342,100 size 24x102
      Visibility <- "Property_1.EstadoSensorMax"
   Rectangle "braco2_2" at 279,101 size 24x102
      Visibility <- "Property_1.ComprimentoXEixo"
   Rectangle "braco" at 154,132 size 55x37
      Visibility <- "Property_1.EstadoSensorMin"
   Rectangle "braco2" at 209,100 size 24x102
      Visibility <- "Property_1.EstadoSensorMin"
*)

(* ===== HMI "HMI_RT_1" =====
system functions are stored by id; their names below are inferred from use

ScreenModuleEditorView "pistao" 640x480
   Button "manual/automatico" at 247,23 size 166x49; TextOn 'MANUAL'; TextOff 'AUTOMATICO'
      on Click: InvertBit("Property_1.ModoControle")
      ProcessValue <- "Property_1.ModoControle"
   Rectangle "braco_1" at 154,132 size 188x37
      Visibility <- "Property_1.EstadoSensorMax"
   Circle "extendido" at 313,217 size 53x53
      Appearance <- "Property_1.EstadoSensorMax"
   Circle "recolhido" at 180,217 size 53x53
      Appearance <- "Property_1.EstadoSensorMin"
   Rectangle "braco_2" at 153,132 size 126x37
      Visibility <- "Property_1.ComprimentoXEixo"
   IOField "nome_pistao" at 31,26 size 188x41; FormatPattern ??????????
      ProcessValue <- "Property_1.NomeCilindro"
   Button "OFF" at 91,291 size 92x45; TextOff 'OFF'
      ObjectEnable <- "Property_1.ModoControle"
      Appearance <- "Property_1.EstadoCilindro"
   Button "ON" at 275,290 size 92x45; TextOff 'ON'
      ObjectEnable <- "Property_1.ModoControle"
      Appearance <- "Property_1.EstadoCilindro"
   Rectangle "braco2_1" at 342,100 size 24x102
      Visibility <- "Property_1.EstadoSensorMax"
   Rectangle "braco2_2" at 279,101 size 24x102
      Visibility <- "Property_1.ComprimentoXEixo"
   Rectangle "braco" at 154,132 size 55x37
      Visibility <- "Property_1.EstadoSensorMin"
   Rectangle "braco2" at 209,100 size 24x102
      Visibility <- "Property_1.EstadoSensorMin"
*)

(* ===== HMI "HMI_RT_1" =====
system functions are stored by id; their names below are inferred from use

HMI tags "Default tag table"
   "ManualEnable" : Bool, internal   // Se on, habilita modo manual do motor
   "MotorState" : Bool, internal   // Se on, motor ligado

ScreenModuleEditorView "motor" 640x480
   Circle "armaduraMotor" at 83,97 size 139x139
      Appearance <- "MotorState"
   Button "BtEnableMotor" at 14,19 size 80x60; TextOff 'Text'
      on Click: InvertBit("ManualEnable")
   Button "BtOnMotor" at 114,19 size 80x60; TextOff 'ON'
      on Click: SetBit("MotorState")
      ObjectEnable <- "ManualEnable"
      Appearance <- "MotorState"
   Button "BtOffMotor" at 211,19 size 80x60; TextOff 'OFF'
      on Click: ResetBit("MotorState")
      ObjectEnable <- "ManualEnable"
      Appearance <- "MotorState"
*)